TYPE DUT_USB_Eingang :
STRUCT
	E1		AT %I* : BOOL;
	E2		AT %I* : BOOL;
	E3		AT %I* : BOOL;
	E4		AT %I* : BOOL;
	E5		AT %I* : BOOL;
	E6		AT %I* : BOOL;
	E7		AT %I* : BOOL;
	E8		AT %I* : BOOL;
END_STRUCT
END_TYPE

(* stored: Version 1.1.0.1
   DUT DUT_USB_Eingang: Id {5a400bd8-3542-4832-b336-76e93b70d38d} *)
